// The runner's record of one test: its verdict, its counts, its clock and its
// deadline. One per registered test, owned by the suite.
//
// Written through TestVerdict, read by the reporters. It holds no assertion logic
// and no comparison logic - mixing those in is what takes an object past 673
// lines and made it impossible to test any part of it in isolation.
//
// It holds no detailed report either. Individual checks are streamed to
// I_TestDetailSink as they are recorded; only what the 80-character summary needs
// is kept here, and it is composed once at completion rather than on every check.
// A test with 40 passing checks composes one line and stores nothing per check.
FUNCTION_BLOCK TestJournal
VAR
	_Label		   : T_MaxString;
	_Location	   : T_MaxString;
	_Status		   : E_TestStatus;
	_Kind		   : E_FailureKind;

	_StepLabel	   : T_MaxString;
	// The first failure is kept, not the last. A later failure is usually a
	// consequence of the first, and the first is what the reader must fix.
	_FailDiagnostic : T_MaxString;
	_FailMessage   : T_MaxString;
	_FailStep	   : T_MaxString;

	_Summary	   : T_MaxString;

	_PassCount	   : UDINT;
	_FailCount	   : UDINT;
	_ElapsedCycles : UDINT;
	_IsFirstCycle  : BOOL;

	// All three phases. Only Body is enforced here - the runner bounds the other
	// two, which run outside the span this object measures.
	_Budgets	   : ST_TestBudgets;

	_Stopwatch	   : TestStopwatch;
END_VAR

(*
	No cyclic body. The suite calls Tick once per scan for the active test; every
	other entry point is driven by a recorded check.
*)

// Suite-wide budgets, applied to every phase and unit the test did not claim for
// itself at registration.
//
// Each unit is tracked separately on purpose. A test naming its own wall-clock
// budget still inherits the suite's scan budget, and the reverse. A single
// 'overridden' flag would break exactly that case and nothing else would notice.
//
// Called once, when the run starts. The defaults are not re-applied on a re-run:
// what a test claimed at registration it keeps.
METHOD ApplyDefaults
VAR_INPUT
	Defaults : ST_TestBudgets;
END_VAR
IF NOT _Budgets.Setup.IsCyclesSet THEN
	_Budgets.Setup.Cycles := Defaults.Setup.Cycles;
END_IF
IF NOT _Budgets.Setup.IsTimeoutSet THEN
	_Budgets.Setup.Timeout := Defaults.Setup.Timeout;
END_IF

IF NOT _Budgets.Body.IsCyclesSet THEN
	_Budgets.Body.Cycles := Defaults.Body.Cycles;
END_IF
IF NOT _Budgets.Body.IsTimeoutSet THEN
	_Budgets.Body.Timeout := Defaults.Body.Timeout;
END_IF

IF NOT _Budgets.Teardown.IsCyclesSet THEN
	_Budgets.Teardown.Cycles := Defaults.Teardown.Cycles;
END_IF
IF NOT _Budgets.Teardown.IsTimeoutSet THEN
	_Budgets.Teardown.Timeout := Defaults.Teardown.Timeout;
END_IF
END_METHOD

// Passed and failed together.
PROPERTY AssertionCount : UDINT
GET
AssertionCount := _PassCount + _FailCount;
END_GET
END_PROPERTY

// Called once by the suite when this test becomes the active one.
METHOD Begin
VAR_INPUT
	Label	 : T_MaxString;
	Location : T_MaxString;
END_VAR
THIS^.Reset();
_Label		  := Label;
_Location	  := Location;
_Status		  := E_TestStatus.Running;
_IsFirstCycle := TRUE;
_Stopwatch.Start();
END_METHOD

// The resolved budgets for all three phases, read by the runner to arm the setup
// and teardown deadlines. Valid once the run has started and ApplyDefaults has
// been called.
PROPERTY Budgets : ST_TestBudgets
GET
Budgets := _Budgets;
END_GET
END_PROPERTY

PROPERTY ElapsedCycles : UDINT
GET
ElapsedCycles := _ElapsedCycles;
END_GET
END_PROPERTY

// Seconds elapsed for this test. Backs I_TestTiming.ElapsedTime.
PROPERTY ElapsedTime : LREAL
GET
ElapsedTime := _Stopwatch.Elapsed;
END_GET
END_PROPERTY

// Terminal. Composes the summary once and stops the clock.
//
// Named Finish, not Complete: a status word as a method name reads as a question,
// and
// Complete collides with IsComplete on the status interface.
//
// A Passed verdict with no recorded check becomes Errored: a body that checked
// nothing usually means a branch never ran, and reporting that green is a silent
// false pass.
METHOD Finish
VAR_INPUT
	Status : E_TestStatus;
END_VAR
IF _Status <> E_TestStatus.Running THEN
	RETURN;
END_IF

_Stopwatch.Stop();

IF _FailCount > 0 THEN
	_Status := SEL(_Kind = E_FailureKind.Environment, E_TestStatus.Failed, E_TestStatus.Errored);
ELSIF (Status = E_TestStatus.Passed) AND (_PassCount = 0) THEN
	_Status			 := E_TestStatus.Errored;
	_Kind			 := E_FailureKind.Environment;
	_FailDiagnostic := 'completed without recording a check';
ELSE
	_Status := Status;
END_IF

_Summary := TestSummaryLine(StepLabel  := _FailStep,
							Diagnostic := _FailDiagnostic,
							Message	   := _FailMessage);
END_METHOD

PROPERTY IsFirstCycle : BOOL
GET
IsFirstCycle := _IsFirstCycle;
END_GET
END_PROPERTY

PROPERTY Kind : E_FailureKind
GET
Kind := _Kind;
END_GET
END_PROPERTY

PROPERTY Label : T_MaxString
GET
Label := _Label;
END_GET
END_PROPERTY

PROPERTY Location : T_MaxString
GET
Location := _Location;
END_GET
SET
// R13: validated before storing. An instance path is a diagnostic, so a bad one
// should read as "not supplied" rather than send the reader somewhere that does
// not exist.
//
// Length is the only check available: T_MaxString truncates silently at 255, and a
// path cut mid-segment names a place that is not there. An empty classname is
// honest; a wrong one is worse than none.
IF LEN(Location) >= 255 THEN
	_Location := '';
	RETURN;
END_IF

_Location := Location;
END_SET
END_PROPERTY

// Terminal without running. A skipped test is not a failure and must not turn a
// build red.
METHOD MarkSkipped
THIS^.Reset();
_Status := E_TestStatus.Skipped;
END_METHOD

// One failed check. The verdict becomes Failed and cannot return to Passed.
//
// Only the FIRST failure's text is kept for the summary. A later failure is
// usually downstream of the first, and the summary has room for one. Every
// failure, including the discarded ones, still reaches the detail sink.
METHOD RecordFailure
VAR_INPUT
	Kind	   : E_FailureKind;
	Diagnostic : T_MaxString;
	Message	   : T_MaxString;
END_VAR
_FailCount := _FailCount + 1;

IF _FailCount = 1 THEN
	_Kind			 := Kind;
	_FailDiagnostic := Diagnostic;
	_FailMessage	 := Message;
	_FailStep		 := _StepLabel;
END_IF
END_METHOD

// One satisfied check. Nothing but the count: the check's own text goes straight
// to the detail sink and is never held here.
METHOD RecordPass
_PassCount := _PassCount + 1;
END_METHOD

// Back to as-declared, keeping the label and location. Used by a re-run: the
// registered set is not redefined, only re-executed.
METHOD Reset
_Status			 := E_TestStatus.NotStarted;
_Kind			 := E_FailureKind.None;
_StepLabel		 := '';
_FailDiagnostic := '';
_FailMessage	 := '';
_FailStep		 := '';
_Summary		 := '';
_PassCount		 := 0;
_FailCount		 := 0;
_ElapsedCycles	 := 0;
_IsFirstCycle	 := FALSE;
_Stopwatch.Reset();
END_METHOD

// What this test claimed for itself at registration. Whatever it did not claim is
// filled in from the suite defaults when the run starts.
//
// Set once, before anything runs, and never while a phase is in progress. A
// deadline that can move during the work it bounds stops detecting the thing it
// exists for.
METHOD SetBudgets
VAR_INPUT
	Budgets : ST_TestBudgets;
END_VAR
_Budgets := Budgets;
END_METHOD

// Purely diagnostic. Its value is captured with the first failure, so a later
// step cannot relabel an earlier one.
METHOD SetStep
VAR_INPUT
	Label : T_MaxString;
END_VAR
_StepLabel := Label;
END_METHOD

PROPERTY Status : E_TestStatus
GET
Status := _Status;
END_GET
END_PROPERTY

// The step label currently set, or empty. Read by TestVerdict so a streamed check
// carries the step it ran under, and by a teardown that behaves differently
// depending on how far the test got.
//
// Read-only. SetStep is the only way in.
PROPERTY StepLabel : T_MaxString
GET
StepLabel := _StepLabel;
END_GET
END_PROPERTY

// Composed to fit 80 characters. Empty until the test completes.
PROPERTY Summary : T_MaxString
GET
Summary := _Summary;
END_GET
END_PROPERTY

// Advance one scan. Returns TRUE if a deadline has just expired, in which case
// the suite abandons the test - the verdict is already recorded here.
//
// Called AFTER the test body has run, so a budget of one allows one execution.
// That ordering is also why ElapsedCycles reads N-1 during the body's Nth call:
// the scan in progress has not completed, so it is not counted. A test observing
// its own duration needs one scan more than the duration it observes.
METHOD Tick : BOOL
Tick := FALSE;

IF _Status <> E_TestStatus.Running THEN
	RETURN;
END_IF

// Only the first scan is the first scan.
_IsFirstCycle  := FALSE;
_ElapsedCycles := _ElapsedCycles + 1;

IF (_Budgets.Body.Cycles > 0) AND (_ElapsedCycles >= _Budgets.Body.Cycles) THEN
	THIS^.RecordFailure(
		Kind	   := E_FailureKind.Timeout,
		Diagnostic := TestTimeoutDiagnostic(Phase	 := '',
											Cycles	 := _Budgets.Body.Cycles,
											Timeout	 := _Budgets.Body.Timeout,
											ByCycles := TRUE),
		Message	   := '');
	THIS^.Finish(E_TestStatus.Failed);
	Tick := TRUE;
	RETURN;
END_IF

IF (_Budgets.Body.Timeout > T#0S) AND (_Stopwatch.Elapsed >= (TO_LREAL(TIME_TO_UDINT(_Budgets.Body.Timeout)) / 1000.0)) THEN
	THIS^.RecordFailure(
		Kind	   := E_FailureKind.Timeout,
		Diagnostic := TestTimeoutDiagnostic(Phase	 := '',
											Cycles	 := _Budgets.Body.Cycles,
											Timeout	 := _Budgets.Body.Timeout,
											ByCycles := FALSE),
		Message	   := '');
	THIS^.Finish(E_TestStatus.Failed);
	Tick := TRUE;
END_IF
END_METHOD

END_FUNCTION_BLOCK

(* stored: Version 1.1.0.1, ProductVersion 3.1.4026.18
   POU TestJournal: Id {b8a8cfea-0795-47ac-8e9a-17b3c171c645}, SpecialFunc None
   Method ApplyDefaults: Id {c2a2a252-7e44-4c4d-9fca-ebfd25d57080}
   Property AssertionCount: Id {f9e3bac2-0fd4-459b-8f72-4b199d9eb389}
   Get Get: Id {d1a3ae9d-4e6c-4fbe-a85f-2acd965b3e8f}
   Method Begin: Id {7d467deb-6e68-4278-b85a-d1ccb586213a}
   Property Budgets: Id {39cfa526-6364-4b14-b960-61d378a96aee}
   Get Get: Id {323275e7-4d1c-40c9-b1b4-0b6cc22d3337}
   Property ElapsedCycles: Id {a734db6d-2f01-4bad-aabf-a0902aec7086}
   Get Get: Id {a3103c5a-712b-4a70-983a-53989c68db56}
   Property ElapsedTime: Id {0403d3c5-dc22-4fc0-b623-f96801bef105}
   Get Get: Id {35f9721c-c669-44cc-9783-c577ab45e725}
   Method Finish: Id {74cb9823-229c-4015-bdd2-73a1478c3f93}
   Property IsFirstCycle: Id {31eba7f5-a511-4659-9363-3ecd682056bf}
   Get Get: Id {9a09ee75-68fb-472b-a918-423b5f38dcf1}
   Property Kind: Id {278b1a6a-212b-474d-80d5-0066a710311e}
   Get Get: Id {a1788759-da60-4cca-879e-7f6e6339741a}
   Property Label: Id {6551f38d-f079-49da-8360-b056cc7c8dbd}
   Get Get: Id {51f284fd-8569-4334-8c44-457622594439}
   Property Location: Id {f4c29500-15d0-4f16-bc6b-be0256259328}
   Get Get: Id {84dfdc95-b83f-445b-a7fa-72d4f6237036}
   Set Set: Id {9e7099ba-7adb-4bcb-bf58-349556ca92cd}
   Method MarkSkipped: Id {6ffe1afd-37d8-4c9f-b5b6-df2986251304}
   Method RecordFailure: Id {8c9ad501-3e04-429f-b5e6-6698564aa084}
   Method RecordPass: Id {3864deed-7cbe-4589-be43-36d6377c64a8}
   Method Reset: Id {c52a6a9c-d80c-46a9-8c9e-03bcdcb9b679}
   Method SetBudgets: Id {662101c2-f10b-4f21-aab8-9e1a19e0e40a}
   Method SetStep: Id {ca4c5efb-3e0f-4df8-9e22-66e642243020}
   Property Status: Id {8522af21-ee18-40b6-be8e-104fc73db02a}
   Get Get: Id {ada9e8d3-31bc-4446-bae0-b04b56937ba7}
   Property StepLabel: Id {b023333c-c6f5-4035-b431-00ab30dfe985}
   Get Get: Id {8be24e4c-9ecf-4ae8-b7b0-ffd54510f060}
   Property Summary: Id {43bacfae-fb64-46ea-a086-d144f21b3922}
   Get Get: Id {77179aa4-0bbe-4bc3-8596-bbba9bc977c9}
   Method Tick: Id {23c9fd8b-4f8a-4a3c-aa08-eb5383729e62} *)
